Fanuc KAREL source: IO0188.KL

-- PROVISIONAL review KL for V940-1; original PC SHA256 ffbfbaa2cceb57e75476ba1b0944853e44a976bb124a2cabf27cc090041bfe40
-- Incomplete behavior may be omitted. Consult companion uncertainty JSON. Do not deploy.
PROGRAM IO0188
%NOLOCKGROUP
-- UNRESOLVED_LOCAL_POOL 5 cells at code offset 13; source declarations unknown
-- DIRECT_LOCAL_WORD_ACCESS alone does not prove INTEGER, REAL, or BOOLEAN
BEGIN
  -- V9_ZERO_TABLE_METADATA_HINT layout=0001; no indexed target words; source/name/runtime held
  -- V9_ZERO_GLOBAL_LAYOUT_HINT count-one $GROUP table, zero relocation slots, two routine descriptors; executable preamble and source held
  -- UNRESOLVED_PC offsets 0-18; opcodes 2B,2C,7B
  -- UNRESOLVED_PC offsets 23-30; opcodes 9D,23
  -- UNRESOLVED_PC offsets 35-49; opcodes 2E,22,9D,33,35
  -- UNRESOLVED_PC offsets 54-61; opcodes 9D,23
  -- UNRESOLVED_PC offsets 66-77; opcodes 2E,23
  -- UNRESOLVED_PC offsets 82-93; opcodes 9D,19,21,1A
  -- UNRESOLVED_PC offsets 98-102; opcodes 7F
  -- UNRESOLVED_PC offsets 107-111; opcodes 27,AA
  -- UNRESOLVED_PC offsets 116-120; opcodes 7F
END IO0188
